// TIA Portal V20 export
FUNCTION_BLOCK "ErrCom"   // FB303, FBD
{ S7_Optimized_Access := 'FALSE' }
// stored: AutoNumber false, SetENOAutomatically false
   VAR
      Var { S7_SetPoint := 'True'} : "TypeVar";
      T : Array[1..1] of IEC_TIMER;
   END_VAR
   VAR_TEMP
      ComOk : Bool;
      PwrOk : Bool;
      SiOk : Bool;
      EsOk : Bool;
      DoorOk : Bool;
   END_VAR
BEGIN

NETWORK
TITLE = general ok
// communication ok
      AN    "G".errComPc;
      =     #ComOk;

// power supply ok
      AN    "G"."errPs-0F1.1+SGV";
      =     #PwrOk;

// safety ok
      AN    "G".errSafetyModules;
      AN    "Si".aLaserErrFdb;
      AN    "Si".aAdjustmentErrFdb1;
      AN    "Si".aAdjustmentErrFdb2;
      =     #SiOk;

// doors ok
      A     #PwrOk;
      A     #SiOk;
      A     "Si".esInternal;
      =     #DoorOk;

// emergency ok
      A     #PwrOk;
      A     #SiOk;
      =     #EsOk;

REGION Network 2 (SCL): emergency stop

   // emergency stop internal (HMI)
   "ComErr".Err[2000] := #EsOk AND NOT "SI_14SB0/1+HMI" AND NOT "I_14SB0+HMI";
   "ComErr".Err[2001] := #EsOk AND NOT "SI_14SB0/1+HMI" AND NOT "I_14SB1+HMI";
   "ComErr".Err[2002] := #EsOk AND "Si".esInternalAckReq;

   // emergency stop external
   "ComErr".Err[2004] := #EsOk AND NOT "SI_NA_EXT+SGV";
   "ComErr".Err[2005] := #EsOk AND "Si".esExternalAckReq;
END_REGION

REGION Network 3 (SCL): safety doors

   // visual measurement - SGV
   "ComErr".Err[2010] := #DoorOk AND NOT "Si"."SGV-14SS1.TL".sig;
   "ComErr".Err[2011] := #DoorOk AND "Si"."SGV-14SS1.TL".sig AND NOT "Si"."SGV-14SS1.TL".ok;

   "ComErr".Err[2013] := #DoorOk AND NOT "Si"."SGV-14SS1.BL".sig;
   "ComErr".Err[2014] := #DoorOk AND "Si"."SGV-14SS1.BL".sig AND NOT "Si"."SGV-14SS1.BL".ok;

   "ComErr".Err[2016] := #DoorOk AND NOT "Si"."SGV-14SS1.TR".sig;
   "ComErr".Err[2017] := #DoorOk AND "Si"."SGV-14SS1.TR".sig AND NOT "Si"."SGV-14SS1.TR".ok;

   "ComErr".Err[2019] := #DoorOk AND NOT "Si"."SGV-14SS1.BR".sig;
   "ComErr".Err[2020] := #DoorOk AND "Si"."SGV-14SS1.BR".sig AND NOT "Si"."SGV-14SS1.BR".ok;

   // visual measurement - SGX
   "ComErr".Err[2030] := #DoorOk AND NOT "Si"."SGX-14SS1.TL".sig;
   "ComErr".Err[2031] := #DoorOk AND "Si"."SGX-14SS1.TL".sig AND NOT "Si"."SGX-14SS1.TL".ok;

   "ComErr".Err[2033] := #DoorOk AND NOT "Si"."SGX-14SS1.BL".sig;
   "ComErr".Err[2034] := #DoorOk AND "Si"."SGX-14SS1.BL".sig AND NOT "Si"."SGX-14SS1.BL".ok;

   "ComErr".Err[2036] := #DoorOk AND NOT "Si"."SGX-14SS1.TR".sig;
   "ComErr".Err[2037] := #DoorOk AND "Si"."SGX-14SS1.TR".sig AND NOT "Si"."SGX-14SS1.TR".ok;

   "ComErr".Err[2039] := #DoorOk AND NOT "Si"."SGX-14SS1.BR".sig;
   "ComErr".Err[2040] := #DoorOk AND "Si"."SGX-14SS1.BR".sig AND NOT "Si"."SGX-14SS1.BR".ok;
END_REGION

REGION Network 4 (SCL): manual

   // setting mode - SSTL
   "ComErr".Err[2050] := #ComOk AND #PwrOk AND #SiOk AND "Si".esInternal AND "Si".settingModeActive;

   // jog mode - SSTL
   "ComErr".Err[2052] := #ComOk AND #PwrOk AND #SiOk AND "Si".esInternal AND "Si".jogModeActive;

   // air-conditioning off - SSTR
   "ComErr".Err[2054] := #ComOk AND #PwrOk AND "I_0SH1+SSTR";
END_REGION

REGION Network 5 (SCL): safety

   // fault safety modules plc
   "ComErr".Err[2060] := #ComOk AND #PwrOk AND "G".errSafetyModules;

   // areas
   "ComErr".Err[2075] := #ComOk AND #PwrOk AND "SI_NA_EXT+SGV" AND  "SI_14SB0/1+HMI" AND (NOT "Si".esInternal OR NOT "Si".esExternal);

   // monitoring feedback
   "ComErr".Err[2080] := #ComOk AND #PwrOk AND "Si".aLaserErrFdb;
   "ComErr".Err[2081] := #ComOk AND #PwrOk AND "Si".aAdjustmentErrFdb1;
   "ComErr".Err[2082] := #ComOk AND #PwrOk AND "Si".aAdjustmentErrFdb2;
   "ComErr".Err[2083] := #ComOk AND #PwrOk AND  "G".Cfg.xrayActive AND "Si".aXrayErrFdb;
END_REGION

REGION Network 6 (SCL): fault sensor
   "ComErr".Err[2090] := "Sen"."1BTR2+SGV".err;
   "ComErr".Err[2091] := "Sen"."1BTR2+SGX".err;
END_REGION

REGION Network 7 (SCL): fault encoder
   "ComErr".Err[2100] := "Enc"."1BCI1".err;
   "ComErr".Err[2101] := "Enc"."1BCM1".err;
   "ComErr".Err[2102] := "Enc"."1BCO1".err;
END_REGION

REGION Network 8 (SCL): communication
   // fault watchdog
   "ComErr".Err[2110] := "G".errComPc;

   // release infeed
   "ComErr".Err[2111] := "G".errNoReleaseInf;
END_REGION

REGION Network 9 (SCL): fault general

   // power supply
   "ComErr".Err[2120] := "G"."errPs-0F1.1+SGV";

   // air conditioner
   "ComErr".Err[2121] := "G"."errAc-0E1+SGV";
   "ComErr".Err[2122] := "G"."errAc-0E2+SGX";
   "ComErr".Err[2123] := "G"."errAc-0E1.1+SGV";

   // err version
   "ComErr".Err[2125] := "G".errVersion;
END_REGION

REGION Network 10 (SCL): off information
   "ComErr".Err[2140] := "G".adjScannerOff;
   "ComErr".Err[2141] := "G".adjTopOff;
   "ComErr".Err[2142] := "G".adjLeftOff;
   "ComErr".Err[2143] := "G".adjRightOff;
   "ComErr".Err[2144] := "G".air1Off;
   "ComErr".Err[2145] := "G".air2Off;
   "ComErr".Err[2146] := "G".airXrayOff;
   "ComErr".Err[2147] := "G".airDehOff;
END_REGION

REGION Network 11 (SCL): fault adjustment

   // adjustment scannerhousing (-8M1.B+SGV)
   "ComErr".Err[2150] := "ComSd".Data.Scanner.Err;
   "ComErr".Err[2151] := "Enc"."8B1.B".err;
   "ComErr".Err[2152] := "Sen"."8S1.B".err;
   "ComErr".Err[2153] := "Sen"."8S2.B".err;
   "ComErr".Err[2154] := "Si".aAdjustment AND NOT "ComSd".Data.Scanner.refRun AND NOT "ComSd".Data.Scanner.refOk;
   "ComErr".Err[2155] := "Si".aAdjustment AND "ComSd".Data.Scanner.refRun;
   "ComErr".Err[2156] := "Si".aAdjustment AND "AdjScanner_DB".Cmd.auto AND NOT"ComSd".Data.Scanner.PosOk;
   "ComErr".Err[2157] := "Si".aAdjustment AND "ComRd".Data.Scanner.ManModeActive;

   // adjustment metering bar top (-8M1.T+SGV)
   "ComErr".Err[2160] := "ComSd".Data.Top.Err;
   "ComErr".Err[2161] := "ComSd".Data.Top.ErrEnc;
   "ComErr".Err[2162] := "Sen"."8S1.T".err;
   "ComErr".Err[2163] := "Sen"."8S2.T".err;
   "ComErr".Err[2164] := "Si".aAdjustment AND NOT "ComSd".Data.Top.refRun AND NOT "ComSd".Data.Top.refOk;
   "ComErr".Err[2165] := "Si".aAdjustment AND "ComSd".Data.Top.refRun;
   "ComErr".Err[2166] := "Si".aAdjustment AND "AdjTop_DB".Cmd.auto AND ((NOT "G".Cfg.adjTopActiveLinMot AND "Enc"."8BC1.T".notInPos) OR ("G".Cfg.adjTopActiveLinMot AND "Enc"."8U1.T".notInPos));
   "ComErr".Err[2167] := "Si".aAdjustment AND "ComRd".Data.Top.ManModeActive;

   // adjustment metering bar left (-8M1.L+SGV)
   "ComErr".Err[2170] := "ComSd".Data.Left.Err;
   "ComErr".Err[2171] := "ComSd".Data.Left.ErrEnc;
   "ComErr".Err[2172] := "Sen"."8S1.L".err;
   "ComErr".Err[2173] := "Sen"."8S2.L".err;
   "ComErr".Err[2174] := "Si".aAdjustment AND NOT "ComSd".Data.Left.refRun AND NOT "ComSd".Data.Left.refOk;
   "ComErr".Err[2175] := "Si".aAdjustment AND "ComSd".Data.Left.refRun;
   "ComErr".Err[2176] := "Si".aAdjustment AND "AdjLeft_DB".Cmd.auto AND ((NOT "G".Cfg.adjLeftActiveLinMot AND "Enc"."8BC1.L".notInPos) OR ("G".Cfg.adjLeftActiveLinMot AND "Enc"."8U1.L".notInPos));
   "ComErr".Err[2177] := "Si".aAdjustment AND "ComRd".Data.Left.ManModeActive;

   // adjustment metering bar right (-8M1.R+SGV)
   "ComErr".Err[2180] := "ComSd".Data.Right.Err;
   "ComErr".Err[2181] := "ComSd".Data.Right.ErrEnc;
   "ComErr".Err[2182] := "Sen"."8S1.R".err;
   "ComErr".Err[2183] := "Sen"."8S2.R".err;
   "ComErr".Err[2184] := "Si".aAdjustment AND NOT "ComSd".Data.Right.refRun AND NOT "ComSd".Data.Right.refOk;
   "ComErr".Err[2185] := "Si".aAdjustment AND "ComSd".Data.Right.refRun;
   "ComErr".Err[2186] := "Si".aAdjustment AND "AdjRight_DB".Cmd.auto AND ((NOT "G".Cfg.adjRightActiveLinMot AND "Enc"."8BC1.R".notInPos) OR ("G".Cfg.adjRightActiveLinMot AND "Enc"."8U1.R".notInPos));
   "ComErr".Err[2187] := "Si".aAdjustment AND "ComRd".Data.Right.ManModeActive;

   // sensor for random adjustment
   "ComErr".Err[2190] := "Sen"."8B1".err AND "G".Cfg.adjTopActiveLinMot;
   "ComErr".Err[2191] := "Sen"."8B2".err AND "G".Cfg.adjLeftActiveLinMot;
   "ComErr".Err[2192] := "Sen"."8B3".err AND "G".Cfg.adjRightActiveLinMot;
END_REGION

REGION Network 12 (SCL): fault profinet

   // fault profinet
   "ComErr".Err[2200] := "Diag_DB".IoDataSys1.devices[1].error AND "G".Cfg.adjTopActiveLinMot;
   "ComErr".Err[2201] := "Diag_DB".IoDataSys1.devices[2].error AND "G".Cfg.adjLeftActiveLinMot;
   "ComErr".Err[2202] := "Diag_DB".IoDataSys1.devices[3].error AND "G".Cfg.adjRightActiveLinMot;
END_REGION
END_FUNCTION_BLOCK
